PROGRAM MAIN
VAR
END_VAR

END_PROGRAM

(* stored: Version 1.1.0.1
   POU MAIN: Id {6b994720-61f3-4a48-9fb0-583e97ad6953}, SpecialFunc None *)
